FUNCTION_BLOCK ModuleCollection_Mockup EXTENDS ModuleCollection<ApplicationBaseParameter.MaxCountInCollections>
VAR
END_VAR

METHOD GetInterfaceById : I_Module
VAR_INPUT
	Id : UDINT;
END_VAR

VAR
	Module : I_Module;
END_VAR
//__QUERYINTERFACE(Modules.GetItemById(Id), Module);

//GetInterfaceById := Module;
END_METHOD

END_FUNCTION_BLOCK

(* stored: Version 1.1.0.1, ProductVersion 3.1.4026.18
   POU ModuleCollection_Mockup: Id {6f9414de-30fb-4e1d-920f-ac583ffa662b}, SpecialFunc None
   Method GetInterfaceById: Id {77e52968-38b0-4b74-8071-d8ef2857a71e} *)
